% RSLogix 500 project project5.RSS, saved by version 8.30.00.16 %
PROJECT "UNTITLED"    % processor: Bul.1763 MicroLogix 1100 Series B %

PROGRAM FILES
  LAD 2 "MAIN"  6 rungs

DATA FILES
  O0 OUTPUT  4 elements
  I1 INPUT  6 elements
  S2 STATUS  66 elements
  B3 BINARY  1 elements
  T4 TIMER  2 elements
  C5 COUNTER  1 elements
  R6 CONTROL  1 elements
  N7 INTEGER  1 elements
  F8 FLOAT  1 elements

LADDER 2 "MAIN"
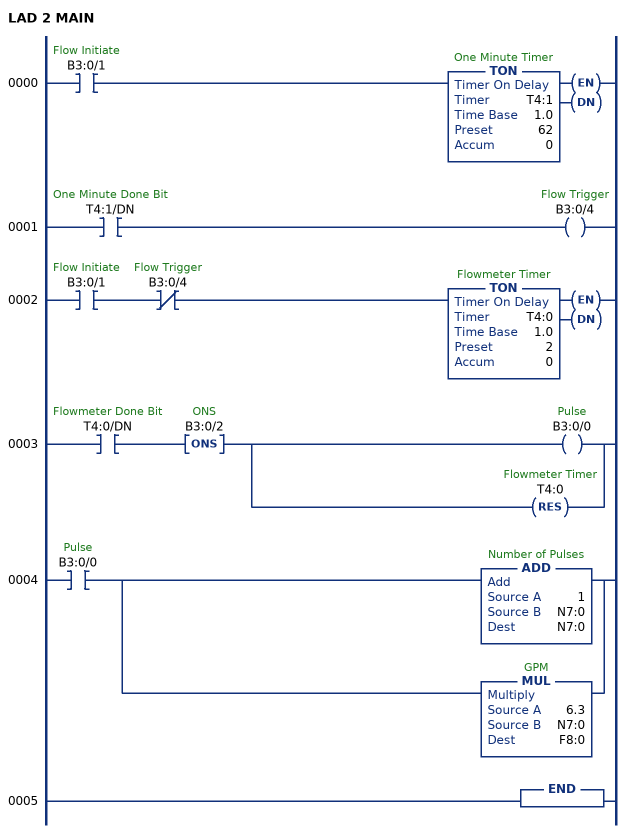
% Rung: 0 %
SOR XIC B3:0/1 TON T4:1 1.0 62 0 EOR
%   B3:0/1  "Flow Initiate" %
%   T4:1  "One Minute Timer" %
% Rung: 1 %
SOR XIC T4:1/DN OTE B3:0/4 EOR
%   T4:1/DN  "One Minute Done Bit" %
%   B3:0/4  "Flow Trigger" %
% Rung: 2 %
SOR XIC B3:0/1 XIO B3:0/4 TON T4:0 1.0 2 0 EOR
%   B3:0/1  "Flow Initiate" %
%   B3:0/4  "Flow Trigger" %
%   T4:0  "Flowmeter Timer" %
% Rung: 3 %
SOR XIC T4:0/DN ONS B3:0/2 BST OTE B3:0/0 NXB RES T4:0 BND EOR
%   T4:0/DN  "Flowmeter Done Bit" %
%   B3:0/2  "ONS" %
%   B3:0/0  "Pulse" %
%   T4:0  "Flowmeter Timer" %
% Rung: 4 %
SOR XIC B3:0/0 BST ADD 1 N7:0 N7:0 NXB MUL 6.3 N7:0 F8:0 BND EOR
%   B3:0/0  "Pulse" %
%   N7:0  "Number of Pulses" %
%   F8:0  "GPM" %
% Rung: 5 %
SOR END EOR

OTHER DOCUMENTED ADDRESSES
  B3:0/3  "ONS"
  B3:0/5  "Timer trigger"
  B3:0/6  "ONS"

DATA TABLE (non-zero values as saved)
DATA T4
% .PRE .ACC %
% T4:0 % 2 0
% T4:1 % 62 0
